FUNCTION_BLOCK Achse1
VAR
	MC_Power_1: MC_POWER;
	MC_Move1: MC_MoveRelative;
END_VAR

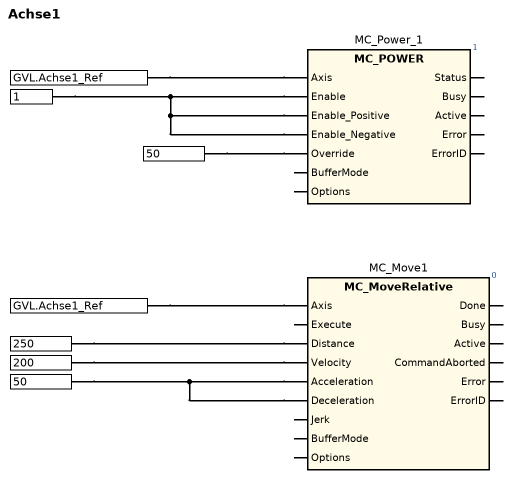
MC_Move1(Axis := GVL.Achse1_Ref, Distance := 250, Velocity := 200, Acceleration := 50, Deceleration := 50); // MC_MoveRelative
MC_Power_1(Axis := GVL.Achse1_Ref, Enable := 1, Enable_Positive := 1, Enable_Negative := 1, Override := 50); // MC_POWER

END_FUNCTION_BLOCK

(* stored: Version 1.1.0.1, ProductVersion 3.1.4024.4
   POU Achse1: Id {3f7df68a-f9b2-4920-934f-1583c9e22ec2}, SpecialFunc None *)
